INTERFACE ITF_BaseDescriptor

END_INTERFACE

(* stored: Version 1.1.0.1
   Itf ITF_BaseDescriptor: Id {ada92c2f-1741-06d9-3083-5dca405ada51} *)
